INTERFACE ITF_TopElement2

END_INTERFACE

(* stored: Version 1.1.0.1, ProductVersion 3.1.4024.15
   Itf ITF_TopElement2: Id {fa26145e-f210-4127-875f-927907ff70c0} *)
